SYSTEM RockerswitchCore
  (* Version 1.0, 2023-01-19, AK124017 *)
  APPLICATION Application
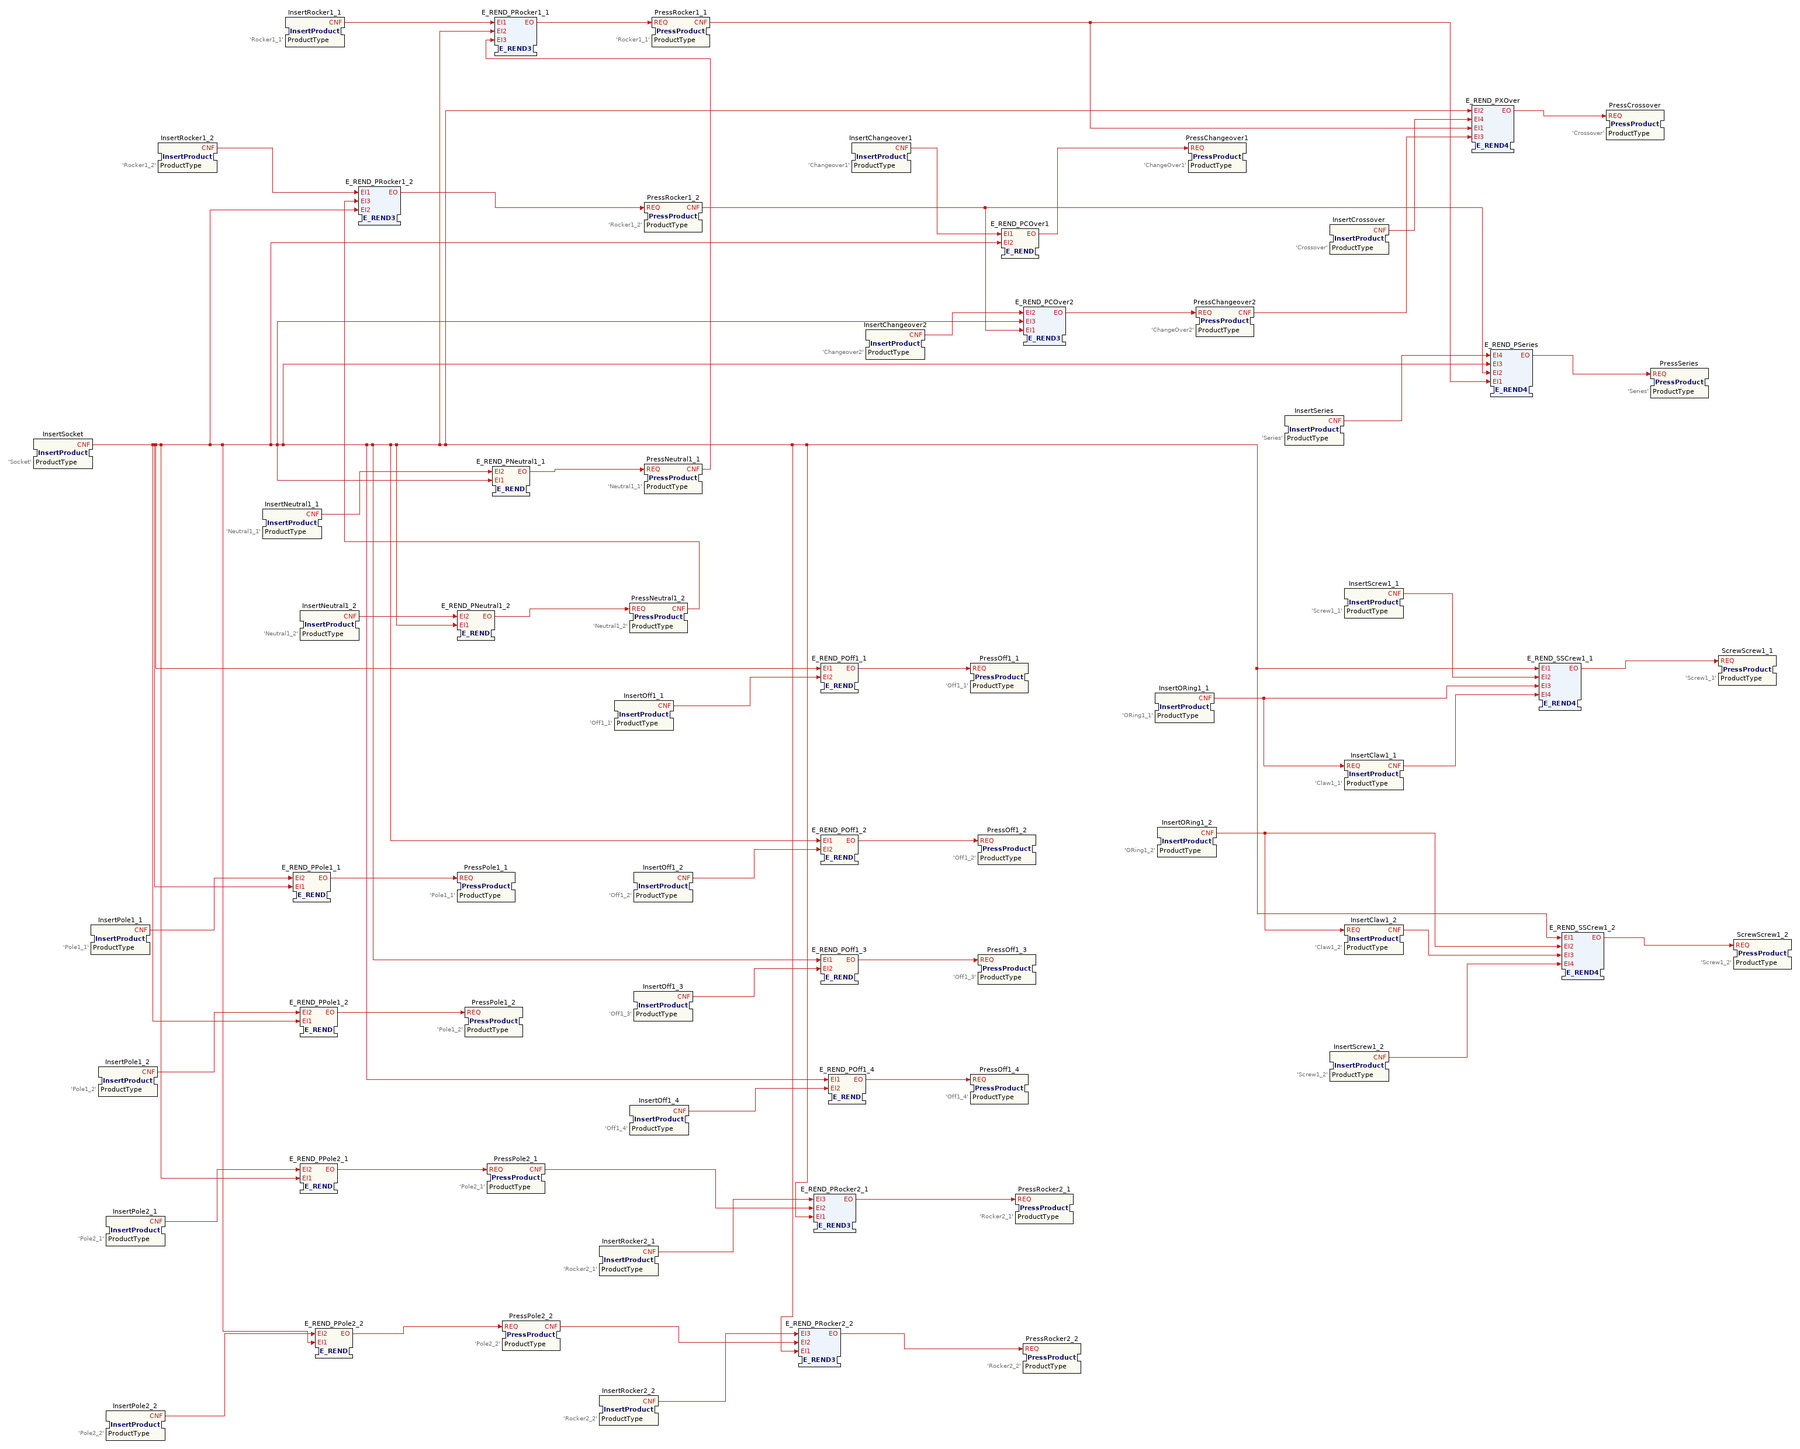
    FBS
      InsertSocket : InsertProduct(ProductType := 'Socket');
      InsertPole1_1 : InsertProduct(ProductType := 'Pole1_1');
      InsertPole1_2 : InsertProduct(ProductType := 'Pole1_2');
      InsertPole2_1 : InsertProduct(ProductType := 'Pole2_1');
      InsertPole2_2 : InsertProduct(ProductType := 'Pole2_2');
      InsertNeutral1_1 : InsertProduct(ProductType := 'Neutral1_1');
      InsertNeutral1_2 : InsertProduct(ProductType := 'Neutral1_2');
      InsertChangeover1 : InsertProduct(ProductType := 'Changeover1');
      InsertChangeover2 : InsertProduct(ProductType := 'Changeover2');
      InsertRocker1_1 : InsertProduct(ProductType := 'Rocker1_1');
      InsertRocker1_2 : InsertProduct(ProductType := 'Rocker1_2');
      InsertOff1_2 : InsertProduct(ProductType := 'Off1_2');
      InsertOff1_3 : InsertProduct(ProductType := 'Off1_3');
      InsertOff1_4 : InsertProduct(ProductType := 'Off1_4');
      InsertCrossover : InsertProduct(ProductType := 'Crossover');
      InsertSeries : InsertProduct(ProductType := 'Series');
      InsertScrew1_1 : InsertProduct(ProductType := 'Screw1_1');
      InsertScrew1_2 : InsertProduct(ProductType := 'Screw1_2');
      InsertORing1_1 : InsertProduct(ProductType := 'ORing1_1');
      InsertORing1_2 : InsertProduct(ProductType := 'ORing1_2');
      InsertClaw1_1 : InsertProduct(ProductType := 'Claw1_1');
      InsertClaw1_2 : InsertProduct(ProductType := 'Claw1_2');
      PressPole1_1 : PressProduct(ProductType := 'Pole1_1');
      PressPole1_2 : PressProduct(ProductType := 'Pole1_2');
      PressPole2_1 : PressProduct(ProductType := 'Pole2_1');
      PressPole2_2 : PressProduct(ProductType := 'Pole2_2');
      PressNeutral1_1 : PressProduct(ProductType := 'Neutral1_1');
      PressNeutral1_2 : PressProduct(ProductType := 'Neutral1_2');
      PressChangeover1 : PressProduct(ProductType := 'ChangeOver1');
      PressChangeover2 : PressProduct(ProductType := 'ChangeOver2');
      PressRocker1_1 : PressProduct(ProductType := 'Rocker1_1');
      PressRocker1_2 : PressProduct(ProductType := 'Rocker1_2');
      PressCrossover : PressProduct(ProductType := 'Crossover');
      PressSeries : PressProduct(ProductType := 'Series');
      ScrewScrew1_1 : PressProduct(ProductType := 'Screw1_1');
      ScrewScrew1_2 : PressProduct(ProductType := 'Screw1_2');
      E_REND_PPole1_1 : E_REND;
      E_REND_PPole1_2 : E_REND;
      E_REND_PPole2_1 : E_REND;
      E_REND_PPole2_2 : E_REND;
      E_REND_PNeutral1_1 : E_REND;
      E_REND_PNeutral1_2 : E_REND;
      E_REND_PCOver1 : E_REND;
      InsertOff1_1 : InsertProduct(ProductType := 'Off1_1');
      InsertRocker2_1 : InsertProduct(ProductType := 'Rocker2_1');
      InsertRocker2_2 : InsertProduct(ProductType := 'Rocker2_2');
      PressRocker2_2 : PressProduct(ProductType := 'Rocker2_2');
      PressRocker2_1 : PressProduct(ProductType := 'Rocker2_1');
      PressOff1_2 : PressProduct(ProductType := 'Off1_2');
      PressOff1_4 : PressProduct(ProductType := 'Off1_4');
      PressOff1_3 : PressProduct(ProductType := 'Off1_3');
      PressOff1_1 : PressProduct(ProductType := 'Off1_1');
      E_REND_POff1_1 : E_REND;
      E_REND_POff1_2 : E_REND;
      E_REND_POff1_3 : E_REND;
      E_REND_POff1_4 : E_REND;
    END_FBS
    SUBAPPS
      E_REND_PCOver2 : E_REND3;
      E_REND_PRocker1_1 : E_REND3;
      E_REND_PRocker1_2 : E_REND3;
      E_REND_PRocker2_2 : E_REND3;
      E_REND_PRocker2_1 : E_REND3;
      E_REND_PXOver : E_REND4;
      E_REND_PSeries : E_REND4;
      E_REND_SSCrew1_1 : E_REND4;
      E_REND_SSCrew1_2 : E_REND4;
    END_SUBAPPS
    EVENT_CONNECTIONS
      InsertORing1_1.CNF TO InsertClaw1_1.REQ;
      InsertORing1_2.CNF TO InsertClaw1_2.REQ;
      InsertPole2_2.CNF TO E_REND_PPole2_2.EI2;
      InsertPole2_1.CNF TO E_REND_PPole2_1.EI2;
      InsertPole1_2.CNF TO E_REND_PPole1_2.EI2;
      InsertPole1_1.CNF TO E_REND_PPole1_1.EI2;
      E_REND_PPole1_1.EO TO PressPole1_1.REQ;
      E_REND_PPole1_2.EO TO PressPole1_2.REQ;
      E_REND_PPole2_1.EO TO PressPole2_1.REQ;
      E_REND_PPole2_2.EO TO PressPole2_2.REQ;
      InsertSocket.CNF TO E_REND_PPole1_1.EI1;
      InsertSocket.CNF TO E_REND_PPole1_2.EI1;
      InsertSocket.CNF TO E_REND_PPole2_1.EI1;
      InsertSocket.CNF TO E_REND_PPole2_2.EI1;
      InsertNeutral1_2.CNF TO E_REND_PNeutral1_2.EI2;
      E_REND_PNeutral1_2.EO TO PressNeutral1_2.REQ;
      InsertSocket.CNF TO E_REND_PNeutral1_2.EI1;
      InsertNeutral1_1.CNF TO E_REND_PNeutral1_1.EI2;
      InsertSocket.CNF TO E_REND_PNeutral1_1.EI1;
      E_REND_PNeutral1_1.EO TO PressNeutral1_1.REQ;
      InsertChangeover1.CNF TO E_REND_PCOver1.EI1;
      InsertSocket.CNF TO E_REND_PCOver1.EI2;
      E_REND_PCOver1.EO TO PressChangeover1.REQ;
      InsertChangeover2.CNF TO E_REND_PCOver2.EI2;
      InsertSocket.CNF TO E_REND_PCOver2.EI3;
      PressRocker1_2.CNF TO E_REND_PCOver2.EI1;
      E_REND_PCOver2.EO TO PressChangeover2.REQ;
      InsertRocker1_1.CNF TO E_REND_PRocker1_1.EI1;
      InsertSocket.CNF TO E_REND_PRocker1_1.EI2;
      PressNeutral1_1.CNF TO E_REND_PRocker1_1.EI3;
      InsertRocker1_2.CNF TO E_REND_PRocker1_2.EI1;
      PressNeutral1_2.CNF TO E_REND_PRocker1_2.EI3;
      InsertSocket.CNF TO E_REND_PRocker1_2.EI2;
      E_REND_PRocker1_1.EO TO PressRocker1_1.REQ;
      E_REND_PRocker1_2.EO TO PressRocker1_2.REQ;
      E_REND_PRocker2_1.EO TO PressRocker2_1.REQ;
      InsertRocker2_2.CNF TO E_REND_PRocker2_2.EI3;
      InsertRocker2_1.CNF TO E_REND_PRocker2_1.EI3;
      E_REND_PRocker2_2.EO TO PressRocker2_2.REQ;
      PressPole2_2.CNF TO E_REND_PRocker2_2.EI2;
      PressPole2_1.CNF TO E_REND_PRocker2_1.EI2;
      InsertSocket.CNF TO E_REND_PRocker2_1.EI1;
      InsertSocket.CNF TO E_REND_PRocker2_2.EI1;
      InsertSocket.CNF TO E_REND_POff1_1.EI1;
      InsertSocket.CNF TO E_REND_POff1_2.EI1;
      InsertSocket.CNF TO E_REND_POff1_3.EI1;
      InsertSocket.CNF TO E_REND_POff1_4.EI1;
      E_REND_POff1_2.EO TO PressOff1_2.REQ;
      E_REND_POff1_3.EO TO PressOff1_3.REQ;
      E_REND_POff1_4.EO TO PressOff1_4.REQ;
      E_REND_POff1_1.EO TO PressOff1_1.REQ;
      InsertOff1_4.CNF TO E_REND_POff1_4.EI2;
      InsertOff1_3.CNF TO E_REND_POff1_3.EI2;
      InsertOff1_2.CNF TO E_REND_POff1_2.EI2;
      InsertOff1_1.CNF TO E_REND_POff1_1.EI2;
      InsertSocket.CNF TO E_REND_PXOver.EI2;
      InsertCrossover.CNF TO E_REND_PXOver.EI4;
      PressRocker1_1.CNF TO E_REND_PXOver.EI1;
      PressChangeover2.CNF TO E_REND_PXOver.EI3;
      E_REND_PXOver.EO TO PressCrossover.REQ;
      E_REND_PSeries.EO TO PressSeries.REQ;
      InsertSeries.CNF TO E_REND_PSeries.EI4;
      InsertSocket.CNF TO E_REND_PSeries.EI3;
      PressRocker1_2.CNF TO E_REND_PSeries.EI2;
      PressRocker1_1.CNF TO E_REND_PSeries.EI1;
      InsertSocket.CNF TO E_REND_SSCrew1_1.EI1;
      InsertSocket.CNF TO E_REND_SSCrew1_2.EI1;
      InsertScrew1_1.CNF TO E_REND_SSCrew1_1.EI2;
      InsertORing1_1.CNF TO E_REND_SSCrew1_1.EI3;
      InsertClaw1_1.CNF TO E_REND_SSCrew1_1.EI4;
      E_REND_SSCrew1_1.EO TO ScrewScrew1_1.REQ;
      InsertORing1_2.CNF TO E_REND_SSCrew1_2.EI2;
      InsertClaw1_2.CNF TO E_REND_SSCrew1_2.EI3;
      InsertScrew1_2.CNF TO E_REND_SSCrew1_2.EI4;
      E_REND_SSCrew1_2.EO TO ScrewScrew1_2.REQ;
    END_CONNECTIONS
  END_APPLICATION
END_SYSTEM
